SUBAPPLICATION Uebung_060 (* für TC-SC also Task Controller Section Control *)
  (* Standard: 61499-2; Description: Copyright (c) 2023 Meisterschulen am Ostbahnhof This program and the accompanying materials are made available under the terms of the Eclipse Public License 2.0 which is available at https://www.eclipse.org/legal/epl-2.0/ SPDX-License-Identifier: EPL-2.0 *)
  (* Version 1.0, 2023-10-23, Franz Höpfinger, Meisterschulen am Ostbahnhof *)
  PACKAGE Uebungen;
  IMPORT TCPool::DE_NUM_DEVICE;
  IMPORT Uebungen::const::TC::DDI::ACTUAL_CONDENSED_WORK_STATE_1_16;
  IMPORT Uebungen::const::TC::DDI::ACTUAL_VOLUME_PER_AREA_APPLICATION_RATE;
  IMPORT Uebungen::const::TC::DDI::ACTUAL_WORK_STATE;
  IMPORT Uebungen::const::TC::DDI::SECTION_CONTROL_STATE;
  IMPORT Uebungen::const::TC::DDI::SETPOINT_CONDENSED_WORK_STATE_1_16;
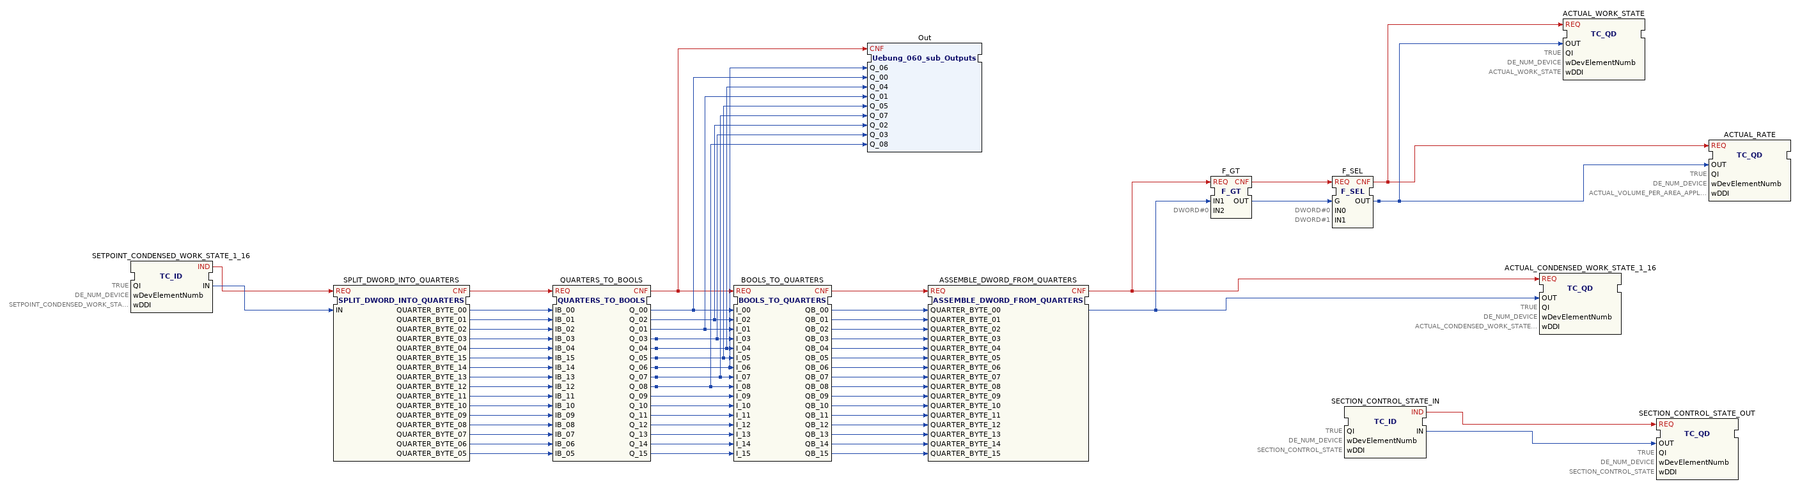
  FBS
    SETPOINT_CONDENSED_WORK_STATE_1_16 : isobus::TC_io::io::TC_ID(QI := TRUE, wDevElementNumb := DE_NUM_DEVICE, wDDI := SETPOINT_CONDENSED_WORK_STATE_1_16);
    SPLIT_DWORD_INTO_QUARTERS : eclipse4diac::utils::splitting::SPLIT_DWORD_INTO_QUARTERS;
    ASSEMBLE_DWORD_FROM_QUARTERS : eclipse4diac::utils::assembling::ASSEMBLE_DWORD_FROM_QUARTERS;
    ACTUAL_CONDENSED_WORK_STATE_1_16 : isobus::TC_io::io::TC_QD(QI := TRUE, wDevElementNumb := DE_NUM_DEVICE, wDDI := ACTUAL_CONDENSED_WORK_STATE_1_16);
    BOOLS_TO_QUARTERS : logiBUS::utils::quarter::BOOLS_TO_QUARTERS;
    QUARTERS_TO_BOOLS : logiBUS::utils::quarter::QUARTERS_TO_BOOLS;
    SECTION_CONTROL_STATE_IN : isobus::TC_io::io::TC_ID(QI := TRUE, wDevElementNumb := DE_NUM_DEVICE, wDDI := SECTION_CONTROL_STATE);
    SECTION_CONTROL_STATE_OUT : isobus::TC_io::io::TC_QD(QI := TRUE, wDevElementNumb := DE_NUM_DEVICE, wDDI := SECTION_CONTROL_STATE);
    ACTUAL_RATE : isobus::TC_io::io::TC_QD(QI := TRUE, wDevElementNumb := DE_NUM_DEVICE, wDDI := ACTUAL_VOLUME_PER_AREA_APPLICATION_RATE);
    ACTUAL_WORK_STATE : isobus::TC_io::io::TC_QD(QI := TRUE, wDevElementNumb := DE_NUM_DEVICE, wDDI := ACTUAL_WORK_STATE);
    F_SEL : iec61131::selection::F_SEL(IN0 := DWORD#0, IN1 := DWORD#1);
    F_GT : iec61131::comparison::F_GT(IN2 := DWORD#0);
  END_FBS
  SUBAPPS
    Out : Uebungen::Uebung_060_sub_Outputs;
  END_SUBAPPS
  EVENT_CONNECTIONS
    SETPOINT_CONDENSED_WORK_STATE_1_16.IND TO SPLIT_DWORD_INTO_QUARTERS.REQ;
    ASSEMBLE_DWORD_FROM_QUARTERS.CNF TO ACTUAL_CONDENSED_WORK_STATE_1_16.REQ;
    BOOLS_TO_QUARTERS.CNF TO ASSEMBLE_DWORD_FROM_QUARTERS.REQ;
    SPLIT_DWORD_INTO_QUARTERS.CNF TO QUARTERS_TO_BOOLS.REQ;
    QUARTERS_TO_BOOLS.CNF TO BOOLS_TO_QUARTERS.REQ;
    QUARTERS_TO_BOOLS.CNF TO Out.CNF;
    SECTION_CONTROL_STATE_IN.IND TO SECTION_CONTROL_STATE_OUT.REQ;
    F_GT.CNF TO F_SEL.REQ;
    ASSEMBLE_DWORD_FROM_QUARTERS.CNF TO F_GT.REQ;
    F_SEL.CNF TO ACTUAL_WORK_STATE.REQ;
    F_SEL.CNF TO ACTUAL_RATE.REQ;
  END_CONNECTIONS
  DATA_CONNECTIONS
    SETPOINT_CONDENSED_WORK_STATE_1_16.IN TO SPLIT_DWORD_INTO_QUARTERS.IN;
    QUARTERS_TO_BOOLS.Q_00 TO BOOLS_TO_QUARTERS.I_00;
    QUARTERS_TO_BOOLS.Q_02 TO BOOLS_TO_QUARTERS.I_02;
    QUARTERS_TO_BOOLS.Q_01 TO BOOLS_TO_QUARTERS.I_01;
    QUARTERS_TO_BOOLS.Q_03 TO BOOLS_TO_QUARTERS.I_03;
    QUARTERS_TO_BOOLS.Q_04 TO BOOLS_TO_QUARTERS.I_04;
    QUARTERS_TO_BOOLS.Q_05 TO BOOLS_TO_QUARTERS.I_05;
    QUARTERS_TO_BOOLS.Q_06 TO BOOLS_TO_QUARTERS.I_06;
    QUARTERS_TO_BOOLS.Q_07 TO BOOLS_TO_QUARTERS.I_07;
    QUARTERS_TO_BOOLS.Q_08 TO BOOLS_TO_QUARTERS.I_08;
    QUARTERS_TO_BOOLS.Q_09 TO BOOLS_TO_QUARTERS.I_09;
    QUARTERS_TO_BOOLS.Q_10 TO BOOLS_TO_QUARTERS.I_10;
    QUARTERS_TO_BOOLS.Q_11 TO BOOLS_TO_QUARTERS.I_11;
    QUARTERS_TO_BOOLS.Q_12 TO BOOLS_TO_QUARTERS.I_12;
    QUARTERS_TO_BOOLS.Q_13 TO BOOLS_TO_QUARTERS.I_13;
    QUARTERS_TO_BOOLS.Q_14 TO BOOLS_TO_QUARTERS.I_14;
    QUARTERS_TO_BOOLS.Q_15 TO BOOLS_TO_QUARTERS.I_15;
    QUARTERS_TO_BOOLS.Q_06 TO Out.Q_06;
    QUARTERS_TO_BOOLS.Q_00 TO Out.Q_00;
    QUARTERS_TO_BOOLS.Q_04 TO Out.Q_04;
    QUARTERS_TO_BOOLS.Q_01 TO Out.Q_01;
    QUARTERS_TO_BOOLS.Q_05 TO Out.Q_05;
    QUARTERS_TO_BOOLS.Q_07 TO Out.Q_07;
    QUARTERS_TO_BOOLS.Q_02 TO Out.Q_02;
    QUARTERS_TO_BOOLS.Q_03 TO Out.Q_03;
    QUARTERS_TO_BOOLS.Q_08 TO Out.Q_08;
    BOOLS_TO_QUARTERS.QB_00 TO ASSEMBLE_DWORD_FROM_QUARTERS.QUARTER_BYTE_00;
    BOOLS_TO_QUARTERS.QB_01 TO ASSEMBLE_DWORD_FROM_QUARTERS.QUARTER_BYTE_01;
    BOOLS_TO_QUARTERS.QB_02 TO ASSEMBLE_DWORD_FROM_QUARTERS.QUARTER_BYTE_02;
    BOOLS_TO_QUARTERS.QB_03 TO ASSEMBLE_DWORD_FROM_QUARTERS.QUARTER_BYTE_03;
    ASSEMBLE_DWORD_FROM_QUARTERS. TO ACTUAL_CONDENSED_WORK_STATE_1_16.OUT;
    BOOLS_TO_QUARTERS.QB_04 TO ASSEMBLE_DWORD_FROM_QUARTERS.QUARTER_BYTE_04;
    BOOLS_TO_QUARTERS.QB_05 TO ASSEMBLE_DWORD_FROM_QUARTERS.QUARTER_BYTE_05;
    BOOLS_TO_QUARTERS.QB_06 TO ASSEMBLE_DWORD_FROM_QUARTERS.QUARTER_BYTE_06;
    BOOLS_TO_QUARTERS.QB_07 TO ASSEMBLE_DWORD_FROM_QUARTERS.QUARTER_BYTE_07;
    BOOLS_TO_QUARTERS.QB_08 TO ASSEMBLE_DWORD_FROM_QUARTERS.QUARTER_BYTE_08;
    BOOLS_TO_QUARTERS.QB_09 TO ASSEMBLE_DWORD_FROM_QUARTERS.QUARTER_BYTE_09;
    BOOLS_TO_QUARTERS.QB_10 TO ASSEMBLE_DWORD_FROM_QUARTERS.QUARTER_BYTE_10;
    BOOLS_TO_QUARTERS.QB_11 TO ASSEMBLE_DWORD_FROM_QUARTERS.QUARTER_BYTE_11;
    BOOLS_TO_QUARTERS.QB_12 TO ASSEMBLE_DWORD_FROM_QUARTERS.QUARTER_BYTE_12;
    BOOLS_TO_QUARTERS.QB_13 TO ASSEMBLE_DWORD_FROM_QUARTERS.QUARTER_BYTE_13;
    BOOLS_TO_QUARTERS.QB_14 TO ASSEMBLE_DWORD_FROM_QUARTERS.QUARTER_BYTE_14;
    BOOLS_TO_QUARTERS.QB_15 TO ASSEMBLE_DWORD_FROM_QUARTERS.QUARTER_BYTE_15;
    SPLIT_DWORD_INTO_QUARTERS.QUARTER_BYTE_00 TO QUARTERS_TO_BOOLS.IB_00;
    SPLIT_DWORD_INTO_QUARTERS.QUARTER_BYTE_01 TO QUARTERS_TO_BOOLS.IB_01;
    SPLIT_DWORD_INTO_QUARTERS.QUARTER_BYTE_02 TO QUARTERS_TO_BOOLS.IB_02;
    SPLIT_DWORD_INTO_QUARTERS.QUARTER_BYTE_03 TO QUARTERS_TO_BOOLS.IB_03;
    SPLIT_DWORD_INTO_QUARTERS.QUARTER_BYTE_04 TO QUARTERS_TO_BOOLS.IB_04;
    SPLIT_DWORD_INTO_QUARTERS.QUARTER_BYTE_15 TO QUARTERS_TO_BOOLS.IB_15;
    SPLIT_DWORD_INTO_QUARTERS.QUARTER_BYTE_14 TO QUARTERS_TO_BOOLS.IB_14;
    SPLIT_DWORD_INTO_QUARTERS.QUARTER_BYTE_13 TO QUARTERS_TO_BOOLS.IB_13;
    SPLIT_DWORD_INTO_QUARTERS.QUARTER_BYTE_12 TO QUARTERS_TO_BOOLS.IB_12;
    SPLIT_DWORD_INTO_QUARTERS.QUARTER_BYTE_11 TO QUARTERS_TO_BOOLS.IB_11;
    SPLIT_DWORD_INTO_QUARTERS.QUARTER_BYTE_10 TO QUARTERS_TO_BOOLS.IB_10;
    SPLIT_DWORD_INTO_QUARTERS.QUARTER_BYTE_09 TO QUARTERS_TO_BOOLS.IB_09;
    SPLIT_DWORD_INTO_QUARTERS.QUARTER_BYTE_08 TO QUARTERS_TO_BOOLS.IB_08;
    SPLIT_DWORD_INTO_QUARTERS.QUARTER_BYTE_07 TO QUARTERS_TO_BOOLS.IB_07;
    SPLIT_DWORD_INTO_QUARTERS.QUARTER_BYTE_06 TO QUARTERS_TO_BOOLS.IB_06;
    SPLIT_DWORD_INTO_QUARTERS.QUARTER_BYTE_05 TO QUARTERS_TO_BOOLS.IB_05;
    SECTION_CONTROL_STATE_IN.IN TO SECTION_CONTROL_STATE_OUT.OUT;
    F_GT.OUT TO F_SEL.G;
    ASSEMBLE_DWORD_FROM_QUARTERS. TO F_GT.IN1;
    F_SEL.OUT TO ACTUAL_RATE.OUT;
    F_SEL.OUT TO ACTUAL_WORK_STATE.OUT;
  END_CONNECTIONS
END_SUBAPPLICATION
